TYPE T_Ctrl_SIf_COS_Cur :
STRUCT
END_STRUCT
END_TYPE

(* stored: Version 1.1.0.1, ProductVersion 3.1.0.19
   DUT T_Ctrl_SIf_COS_Cur: Id {7431ee51-8dc0-43ee-9579-297bb38e79ee} *)
